RoboDK station: Assembly-with-ABB-IRB-2400-16.rdk

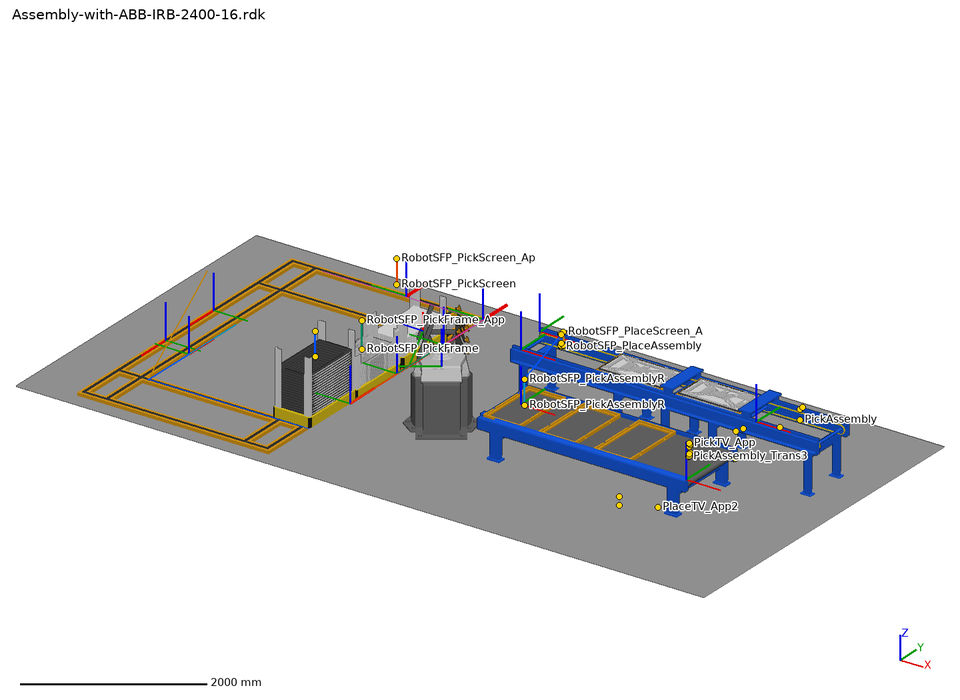
[picture v0: the station drawn from its stored meshes, robots at their saved joint values, targets as dots, program paths as lines]
Station Assembly with ABB IRB 2400/16 (saved by RoboDK 5.6.8). Poses are relative to the parent item; angles as X-Y-Z fixed-axis rotations.
Station parameters (name, value as stored): Assembly, 1, NextAssembly, 1, ScrewCircuit, 1, BuildCircuit, 1, UpFoamDone, 0, RackReady, 0, TAGS, ['Assembly']
  - folder First_Assembly_Station
    - folder Python
      - Python program RackConveyor_Next (listed below)
      - Python program MainConveyor_Next (listed below)
    - folder RobotSFP_Programs
      - folder Gripper1
        - program Gripper1Open (2 instructions, listed below)
        - program Gripper1CloseFrame (2 instructions, listed below)
        - program Gripper1CloseAssemRack (2 instructions, listed below)
        - program Gripper1OpenPartial (2 instructions, listed below)
        - program Gripper1CloseFrontPanel (2 instructions, listed below)
      - folder AssemblyPicks
        - program PickFrontPanel (8 instructions, listed below)
        - program PickScreen (6 instructions, listed below)
        - program PickFrame (8 instructions, listed below)
      - folder PlaceOnAssembly
        - program PlaceFrontPanel (9 instructions, listed below)
        - program PlaceScreen (9 instructions, listed below)
        - program PickAndPlace_AssemRack (14 instructions, listed below)
        - program PlaceFrame (11 instructions, listed below)
      - folder AssemblyProcess
        - program AssemblyTV (6 instructions, listed below)
    - frame MainConveyor Base at (-1580, 450, 650) mm
      - robot MainConveyor: 1 axes
          modified DH rows (alpha deg, a mm, theta deg, d mm): 0, 0, 0, 0 linear
          base shift (0, 0, 0) mm, rotated rx 0 ry 90 rz 0 deg
          joint limits [-200000] to [200000]; home [0]; saved at [0]
        - frame MainConveyorRef at (90, -480, 0) mm
          - object TVAssemblies at (2875, 462, 0) mm, rotated rx 0 ry 0 rz -180 deg, size 1893 x 485 x 64 mm
      - frame MainConveyorRef_Init at (3165, -480, 0) mm
        - object TVAssemblies at (-200, 462, 0) mm, rotated rx 0 ry 0 rz -180 deg, size 1893 x 485 x 64 mm
      - frame RobotSFP_Targets at (-1430, 980, -645) mm, rotated rx 0 ry 0 rz 90 deg
        - frame AssemblyRack_Targets at (0, 1000, 0) mm
          - target RobotSFP_PickAssemblyRack (Cartesian target) at (-2266, -3132, 478) mm, rotated rx 180 ry 0 rz -180 deg; joints [-130.241, 56.24, 97.421, -5.047, -77.391, -90.693] of ABB IRB 2400/16
          - target RobotSFP_PickAssemblyRack_App (Cartesian target) at (-2266, -3132, 790) mm, rotated rx -180 ry 0 rz -180 deg; joints [-130.241, 25.611, 75.665, -5.962, -55.732, -88.432] of ABB IRB 2400/16
          - target RobotSFP_PlaceAssemblyRack (Cartesian target) at (-1226, -2885, 690) mm, rotated rx 180 ry 0 rz -90 deg; joints [-92.609, 47.662, 66.312, -67.815, -58.973, -66.679] of ABB IRB 2400/16
          - target RobotSFP_PlaceAssemblyRack_App (Cartesian target) at (-1226, -2885, 830) mm, rotated rx -180 ry 0 rz -90 deg; joints [-92.609, 38.532, 58.57, -72.434, -56.335, -58.059] of ABB IRB 2400/16
        - frame TvAssembly at (0, 0, -20) mm
          - target RobotSFP_PlaceFrontPanel (Cartesian target) at (-1232.5, -1885.5, 730.48) mm, rotated rx 180 ry 0 rz -90 deg; joints [-92.924, 46.128, 65.422, -68.631, -58.762, -65.657] of ABB IRB 2400/16
          - target RobotSFP_PlaceFrontPanel_App (Cartesian target) at (-1232.5, -1885.5, 863.5) mm, rotated rx -180 ry 0 rz -90 deg; joints [-92.924, 37.534, 57.905, -73.159, -56.297, -57.237] of ABB IRB 2400/16
          - target RobotSFP_PlaceScreen (Cartesian target) at (-1189.8, -1890.5, 709.68) mm, rotated rx 180 ry 0 rz 90 deg; joints [-91.494, 45.247, 62.599, -68.849, -57.154, 117.178] of ABB IRB 2400/16
          - target RobotSFP_PlaceScreen_App (Cartesian target) at (-1189.8, -1890.5, 871.7) mm, rotated rx 180 ry 0 rz 90 deg; joints [-91.494, 35.396, 53.282, -74.906, -54.246, 127.901] of ABB IRB 2400/16
          - target RobotSFP_PlaceFrame (Cartesian target) at (-1219.5, -1885.2, 745.48) mm, rotated rx 180 ry 0 rz -90 deg; joints [-92.315, 45.44, 64.267, -68.683, -58.101, -64.505] of ABB IRB 2400/16
          - target RobotSFP_PlaceFrame_App (Cartesian target) at (-1219.5, -1885.2, 853.5) mm, rotated rx -180 ry 0 rz -90 deg; joints [-92.315, 38.518, 58.189, -72.396, -56.073, -57.678] of ABB IRB 2400/16
      - frame PickAssembly_Targets at (89.8, -480, -648) mm
        - target PickAssembly (Cartesian target) at (3485.2, 228, 693.7) mm, rotated rx -180 ry 0 rz -180 deg; joints [22.371, 48.063, -2.442, 0, 44.379, 112.371]
        - target PickAssembly_App (Cartesian target) at (3485.2, 228, 823.7) mm, rotated rx -180 ry 0 rz -180 deg; joints [22.371, 43.327, -4.321, 0, 50.994, 112.371]
        - target PickAssembly_Trans1 (Cartesian target) at (3525.2, 228, 853.7) mm, rotated rx 180 ry 5 rz 180 deg; joints [21.562, 41.902, -4.058, -5.74, 54.134, 115.007]
        - target PickAssembly_Trans2 (Cartesian target) at (3605.2, -312, 853.7) mm, rotated rx -180 ry 0 rz 80 deg; joints [28.286, 14.78, 41.406, 0, 33.814, 218.286]
        - target PickAssembly_Trans3 (Cartesian target) at (2776, -836.2, 483.7) mm, rotated rx -180 ry 0 rz 90 deg; joints [77.346, 50.715, 13.544, 0, 25.741, 257.346]
      - object Floor at (-100, -970, -650) mm, size 9000 x 4500 x 0 mm, geometry from Floor (2).sld
    - frame ABB IRB 2400/16 Base at (-2010, -770, 600) mm, rotated rx 0 ry 0 rz 125 deg
      - robot ABB IRB 2400/16: 6 axes, payload 16 kg, reach 1550 mm, repeatability 0.03 mm, weight 380 kg
          joint limits [-180, -100, -60, -200, -120, -400] to [180, 110, 65, 200, 120, 400]; home [0, 0, 0, 0, 0, 0]; saved at [-92.609, 38.532, 58.57, -72.434, -56.335, -58.059]
        - frame ToolRobot1 Base at (0, 195, 425) mm, rotated rx -70 ry 0 rz 0 deg
          - robot ToolRobot1: 1 axes
              joint limits [-20] to [200]; home [0]; saved at [26]
        - tool ToolRobot1_TCP_Gripper, TCP at (0, 195, 425) mm, rotated rx -70 ry 0 rz 0 deg
        - tool ToolRobot1_TCP_Cup, TCP at (0, -240, 450) mm, rotated rx 70 ry 0 rz 0 deg
      - target Gripper1Open (Cartesian target) at (1586.9, 365.98, 80) mm, rotated rx 180 ry 0 rz -35 deg; joints [100, -0.574, 0, 0, -0.574, -0.819] of ToolRobot1
      - target Gripper1CloseFrame (Cartesian target) at (858.67, 851.47, -365) mm, rotated rx -180 ry 0 rz -35 deg; joints [-4, 0, 0, 0, 0, 0] of ToolRobot1
      - target Gripper1CloseAssemRack (Cartesian target) at (-703.35, -889.42, -270) mm, rotated rx 180 ry 0 rz 145 deg; joints [26, 0.574, 0, 0, 0.574, 0.819] of ToolRobot1
      - target Gripper1OpenPartial (Cartesian target) at (320.55, -1292.63, -60) mm, rotated rx -180 ry 0 rz -125 deg; joints [50, -0.819, 0, 0, -0.819, 0.574] of ToolRobot1
      - target Gripper1CloseFrontPanel (Cartesian target) at (136.59, 1363.18, -105) mm, rotated rx -180 ry 0 rz -35 deg; joints [41, -0.574, 0, 0, -0.574, -0.819] of ToolRobot1
      - object Robot1_Stand at (0, 0, 0) mm, size 938.8 x 824.6 x 600 mm, geometry from Robot1_Stand.step
    - frame AssemblyRackConveyor Base at (1530, -1260, 440) mm
      - robot AssemblyRackConveyor: 1 axes
          modified DH rows (alpha deg, a mm, theta deg, d mm): 0, 0, 0, 0 linear
          base shift (0, 0, 0) mm, rotated rx 0 ry 90 rz 0 deg
          joint limits [-200000] to [200000]; home [0]; saved at [0]
        - frame AssemblyRackConveyorRef at (0, 0, 0) mm
          - object AssemblyRack at (-1440, 0, 0) mm, size 40 x 853 x 485 mm, geometry from AssemblyRack.step
          - object AssemblyRack at (-720, 0, 0) mm, size 40 x 853 x 485 mm, geometry from AssemblyRack.step
          - object AssemblyRack at (-2160, 0, 0) mm, size 40 x 853 x 485 mm, geometry from AssemblyRack.step
      - frame AssemblyRackConveyorRef_Init at (0, 0, 0) mm
        - object AssemblyRack_Ref at (-1440, 0, 0) mm, size 40 x 853 x 485 mm, geometry from AssemblyRack.step
        - object AssemblyRack_Ref at (-720, 0, 0) mm, size 40 x 853 x 485 mm, geometry from AssemblyRack.step
        - object AssemblyRack_Ref at (-2160, 0, 0) mm, size 40 x 853 x 485 mm, geometry from AssemblyRack.step
      - frame AssemblyRackConveyor_Targets at (0, 0, 0) mm
        - target PlaceAssembly_App1 (Cartesian target) at (509.67, 338.93, 613.53) mm, rotated rx -172.41 ry 0.65 rz 63.37 deg; joints [68.32, -23.6, 57.9, -0.01, 48.08, 275]
        - target PlaceAssembly (Cartesian target) at (-254, 423.8, 43.7) mm, rotated rx -180 ry 0 rz 90 deg; joints [77.346, 50.715, 13.544, 0, 25.741, 257.346]
        - target PlaceAssembly_App2 (Cartesian target) at (-254, 423.8, 153.7) mm, rotated rx 180 ry 0 rz 90 deg; joints [77.346, 45.066, 13.905, -180, -31.029, 77.346]
        - target PlaceBackPanel (Cartesian target) at (-241, 423.9, 86) mm, rotated rx 180 ry 0 rz -90 deg; joints [77.214, 48.026, 14.946, 0, 27.028, 77.214]
        - target PlaceBackPanel_App1 (Cartesian target) at (481.6, 244.34, 613.6) mm, rotated rx 172.37 ry 0 rz -101.17 deg; joints [78.83, -23.59, 57.89, 0, 48.07, 90]
        - target PickTV (Cartesian target) at (-252, 423.9, 65) mm, rotated rx 180 ry 0 rz -90 deg; joints [77.322, 49.521, 13.865, 0, 26.614, 77.322]
        - target PlaceBackPanel_App2 (Cartesian target) at (-241, 423.9, 176) mm, rotated rx 180 ry 0 rz -90 deg; joints [77.214, 43.448, 15.011, 0, 31.541, 77.214]
        - target PickTV_App (Cartesian target) at (-252, 423.9, 195) mm, rotated rx 180 ry 0 rz -90 deg; joints [77.322, 42.97, 13.968, 0, 33.062, 77.322]
        - target PlaceTV_App1 (Cartesian target) at (349, 423.9, 176) mm, rotated rx 180 ry 0 rz -90 deg; joints [66.756, 24.897, 59.615, 0, 5.488, 66.756]
        - target PlaceTV_App2 (Cartesian target) at (349, -1026.1, 176) mm, rotated rx -180 ry 0 rz -90 deg; joints [150.453, 45.871, 9.692, 0, 34.437, 150.453]
        - target PlaceTV (Cartesian target) at (-141, -1045, 72) mm, rotated rx 180 ry 0 rz -90 deg; joints [135.834, 66.25, -25.615, 0, 49.365, 135.834]
        - target PlaceTV_App3 (Cartesian target) at (-141, -1045, 172) mm, rotated rx -180 ry 0 rz -90 deg; joints [135.834, 62.358, -25.443, 0, 53.085, 135.834]
    - program TVAssembly_Main (5 instructions, listed below)
  - folder AVG_On_Rail
    - folder Python
      - Python program Next_RackTarget (listed below)
    - folder TvRack_Programs
      - program TvRack_ToPickUp (5 instructions, listed below)
      - program TvRack_FrontPanel_ToPickUp (4 instructions, listed below)
      - program TvRack_Frame_ToPickUp (4 instructions, listed below)
      - program TvRack_Screen_ToPickUp (4 instructions, listed below)
      - program TvRack_BackToFill (5 instructions, listed below)
      - program TvRack_FrontPanel_ToFill (4 instructions, listed below)
      - program TvRack_Frame_ToFill (4 instructions, listed below)
      - program TvRack_Screen_ToFill (4 instructions, listed below)
    - frame TvRack_Rail at (-3000, 1420, 0) mm, rotated rx 0 ry 0 rz 90 deg
      - robot TvRack_FrontPanel: 2 axes
          modified DH rows (alpha deg, a mm, theta deg, d mm): 0, 0, 0, 0 linear; 90, 0, 0, 0 linear
          base shift (0, 0, 0) mm, rotated rx 0 ry 90 rz 0 deg
          joint limits [-3250, -2100] to [0, 0]; home [0, 0]; saved at [-2480, 0]
        - frame TvRack_FrontPanel_Ref at (0, 0, 0) mm
          - object TVFrontPanel at (-750, 400, 0) mm, rotated rx 0 ry 0 rz 180 deg, size 812.6 x 460.3 x 32.5 mm, geometry from TVFrontCase.step
          - object TVFrontPanel at (-750, 400, 30) mm, rotated rx 0 ry 0 rz 180 deg, size 812.6 x 460.3 x 32.5 mm, geometry from TVFrontCase.step
          - object TVFrontPanel at (-750, 400, 60) mm, rotated rx 0 ry 0 rz 180 deg, size 812.6 x 460.3 x 32.5 mm, geometry from TVFrontCase.step
          - object TVFrontPanel at (-750, 400, 90) mm, rotated rx 0 ry 0 rz 180 deg, size 812.6 x 460.3 x 32.5 mm, geometry from TVFrontCase.step
          - object TVFrontPanel at (-750, 400, 120) mm, rotated rx 0 ry 0 rz 180 deg, size 812.6 x 460.3 x 32.5 mm, geometry from TVFrontCase.step
          - object TVFrontPanel at (-750, 400, 150) mm, rotated rx 0 ry 0 rz 180 deg, size 812.6 x 460.3 x 32.5 mm, geometry from TVFrontCase.step
          - object TVFrontPanel at (-750, 400, 180) mm, rotated rx 0 ry 0 rz 180 deg, size 812.6 x 460.3 x 32.5 mm, geometry from TVFrontCase.step
          - object TVFrontPanel at (-750, 400, 210) mm, rotated rx 0 ry 0 rz 180 deg, size 812.6 x 460.3 x 32.5 mm, geometry from TVFrontCase.step
          - object TVFrontPanel at (-750, 400, 270) mm, rotated rx 0 ry 0 rz 180 deg, size 812.6 x 460.3 x 32.5 mm, geometry from TVFrontCase.step
          - object TVFrontPanel at (-750, 400, 240) mm, rotated rx 0 ry 0 rz 180 deg, size 812.6 x 460.3 x 32.5 mm, geometry from TVFrontCase.step
          - object TVFrontPanel at (-750, 400, 300) mm, rotated rx 0 ry 0 rz 180 deg, size 812.6 x 460.3 x 32.5 mm, geometry from TVFrontCase.step
          - object TVFrontPanel at (-750, 400, 330) mm, rotated rx 0 ry 0 rz 180 deg, size 812.6 x 460.3 x 32.5 mm, geometry from TVFrontCase.step
          - object TVFrontPanel at (-750, 400, 360) mm, rotated rx 0 ry 0 rz 180 deg, size 812.6 x 460.3 x 32.5 mm, geometry from TVFrontCase.step
          - object TVFrontPanel at (-750, 400, 390) mm, rotated rx 0 ry 0 rz 180 deg, size 812.6 x 460.3 x 32.5 mm, geometry from TVFrontCase.step
          - object TVFrontPanel at (-750, 400, 420) mm, rotated rx 0 ry 0 rz 180 deg, size 812.6 x 460.3 x 32.5 mm, geometry from TVFrontCase.step
          - object TVFrontPanel at (-750, 400, 450) mm, rotated rx 0 ry 0 rz 180 deg, size 812.6 x 460.3 x 32.5 mm, geometry from TVFrontCase.step
      - robot TvRack_Frame: 2 axes
          modified DH rows (alpha deg, a mm, theta deg, d mm): 0, 0, 0, 0 linear; 90, 0, 0, 0 linear
          base shift (0, 0, 0) mm, rotated rx 0 ry 90 rz 0 deg
          joint limits [-3250, -2100] to [0, 0]; home [0, 0]; saved at [-1600, 0]
        - frame TvRack_Frame_Ref at (0, 0, 0) mm
          - object TVFrame at (-750, 400, 0) mm, rotated rx 0 ry 0 rz -180 deg, size 786.6 x 406 x 28 mm, geometry from TVFrame.step
          - object TVFrame at (-750, 400, 15) mm, rotated rx 0 ry 0 rz -180 deg, size 786.6 x 406 x 28 mm, geometry from TVFrame.step
          - object TVFrame at (-750, 400, 30) mm, rotated rx 0 ry 0 rz -180 deg, size 786.6 x 406 x 28 mm, geometry from TVFrame.step
          - object TVFrame at (-750, 400, 45) mm, rotated rx 0 ry 0 rz -180 deg, size 786.6 x 406 x 28 mm, geometry from TVFrame.step
          - object TVFrame at (-750, 400, 60) mm, rotated rx 0 ry 0 rz -180 deg, size 786.6 x 406 x 28 mm, geometry from TVFrame.step
          - object TVFrame at (-750, 400, 75) mm, rotated rx 0 ry 0 rz -180 deg, size 786.6 x 406 x 28 mm, geometry from TVFrame.step
          - object TVFrame at (-750, 400, 90) mm, rotated rx 0 ry 0 rz -180 deg, size 786.6 x 406 x 28 mm, geometry from TVFrame.step
          - object TVFrame at (-750, 400, 105) mm, rotated rx 0 ry 0 rz -180 deg, size 786.6 x 406 x 28 mm, geometry from TVFrame.step
          - object TVFrame at (-750, 400, 120) mm, rotated rx 0 ry 0 rz -180 deg, size 786.6 x 406 x 28 mm, geometry from TVFrame.step
          - object TVFrame at (-750, 400, 135) mm, rotated rx 0 ry 0 rz -180 deg, size 786.6 x 406 x 28 mm, geometry from TVFrame.step
          - object TVFrame at (-750, 400, 225) mm, rotated rx 0 ry 0 rz -180 deg, size 786.6 x 406 x 28 mm, geometry from TVFrame.step
          - object TVFrame at (-750, 400, 210) mm, rotated rx 0 ry 0 rz -180 deg, size 786.6 x 406 x 28 mm, geometry from TVFrame.step
          - object TVFrame at (-750, 400, 195) mm, rotated rx 0 ry 0 rz -180 deg, size 786.6 x 406 x 28 mm, geometry from TVFrame.step
          - object TVFrame at (-750, 400, 180) mm, rotated rx 0 ry 0 rz -180 deg, size 786.6 x 406 x 28 mm, geometry from TVFrame.step
          - object TVFrame at (-750, 400, 165) mm, rotated rx 0 ry 0 rz -180 deg, size 786.6 x 406 x 28 mm, geometry from TVFrame.step
          - object TVFrame at (-750, 400, 150) mm, rotated rx 0 ry 0 rz -180 deg, size 786.6 x 406 x 28 mm, geometry from TVFrame.step
      - robot TvRack_Screen: 2 axes
          modified DH rows (alpha deg, a mm, theta deg, d mm): 0, 0, 0, 0 linear; 90, 0, 0, 0 linear
          base shift (0, 0, 0) mm, rotated rx 0 ry 90 rz 0 deg
          joint limits [-3250, -2100] to [0, 0]; home [0, 0]; saved at [-730, 0]
        - frame TvRack_Screen_Ref at (0, 0, 0) mm
          - object TVScreen at (0, 0, 0) mm, size 776.6 x 396 x 12 mm, geometry from TVScreen.step
          - object TVScreen at (0, 0, 12) mm, size 776.6 x 396 x 12 mm, geometry from TVScreen.step
          - object TVScreen at (0, 0, 24) mm, size 776.6 x 396 x 12 mm, geometry from TVScreen.step
          - object TVScreen at (0, 0, 36) mm, size 776.6 x 396 x 12 mm, geometry from TVScreen.step
          - object TVScreen at (0, 0, 48) mm, size 776.6 x 396 x 12 mm, geometry from TVScreen.step
          - object TVScreen at (0, 0, 60) mm, size 776.6 x 396 x 12 mm, geometry from TVScreen.step
          - object TVScreen at (0, 0, 72) mm, size 776.6 x 396 x 12 mm, geometry from TVScreen.step
          - object TVScreen at (0, 0, 84) mm, size 776.6 x 396 x 12 mm, geometry from TVScreen.step
          - object TVScreen at (0, 0, 96) mm, size 776.6 x 396 x 12 mm, geometry from TVScreen.step
          - object TVScreen at (0, 0, 108) mm, size 776.6 x 396 x 12 mm, geometry from TVScreen.step
          - object TVScreen at (0, 0, 120) mm, size 776.6 x 396 x 12 mm, geometry from TVScreen.step
          - object TVScreen at (0, 0, 132) mm, size 776.6 x 396 x 12 mm, geometry from TVScreen.step
          - object TVScreen at (0, 0, 144) mm, size 776.6 x 396 x 12 mm, geometry from TVScreen.step
          - object TVScreen at (0, 0, 180) mm, size 776.6 x 396 x 12 mm, geometry from TVScreen.step
          - object TVScreen at (0, 0, 168) mm, size 776.6 x 396 x 12 mm, geometry from TVScreen.step
          - object TVScreen at (0, 0, 156) mm, size 776.6 x 396 x 12 mm, geometry from TVScreen.step
      - frame TvRack_FrontPanel_Init at (-1460, 2500, 0) mm, rotated rx 0 ry 0 rz 180 deg
        - object TVFrontPanel_Ref at (0, 0, 0) mm, size 812.6 x 460.3 x 32.5 mm, geometry from TVFrontCase.step
        - object TVFrontPanel_Ref at (0, 0, 30) mm, size 812.6 x 460.3 x 32.5 mm, geometry from TVFrontCase.step
        - object TVFrontPanel_Ref at (0, 0, 60) mm, size 812.6 x 460.3 x 32.5 mm, geometry from TVFrontCase.step
        - object TVFrontPanel_Ref at (0, 0, 90) mm, size 812.6 x 460.3 x 32.5 mm, geometry from TVFrontCase.step
        - object TVFrontPanel_Ref at (0, 0, 120) mm, size 812.6 x 460.3 x 32.5 mm, geometry from TVFrontCase.step
        - object TVFrontPanel_Ref at (0, 0, 150) mm, size 812.6 x 460.3 x 32.5 mm, geometry from TVFrontCase.step
        - object TVFrontPanel_Ref at (0, 0, 180) mm, size 812.6 x 460.3 x 32.5 mm, geometry from TVFrontCase.step
        - object TVFrontPanel_Ref at (0, 0, 210) mm, size 812.6 x 460.3 x 32.5 mm, geometry from TVFrontCase.step
        - object TVFrontPanel_Ref at (0, 0, 270) mm, size 812.6 x 460.3 x 32.5 mm, geometry from TVFrontCase.step
        - object TVFrontPanel_Ref at (0, 0, 240) mm, size 812.6 x 460.3 x 32.5 mm, geometry from TVFrontCase.step
        - object TVFrontPanel_Ref at (0, 0, 300) mm, size 812.6 x 460.3 x 32.5 mm, geometry from TVFrontCase.step
        - object TVFrontPanel_Ref at (0, 0, 330) mm, size 812.6 x 460.3 x 32.5 mm, geometry from TVFrontCase.step
        - object TVFrontPanel_Ref at (0, 0, 360) mm, size 812.6 x 460.3 x 32.5 mm, geometry from TVFrontCase.step
        - object TVFrontPanel_Ref at (0, 0, 390) mm, size 812.6 x 460.3 x 32.5 mm, geometry from TVFrontCase.step
        - object TVFrontPanel_Ref at (0, 0, 420) mm, size 812.6 x 460.3 x 32.5 mm, geometry from TVFrontCase.step
        - object TVFrontPanel_Ref at (0, 0, 450) mm, size 812.6 x 460.3 x 32.5 mm, geometry from TVFrontCase.step
      - frame TvRack_Frame_Init at (-2350, 2500, 0) mm, rotated rx 0 ry 0 rz -180 deg
        - object TVFrame_Ref at (0, 0, 0) mm, size 786.6 x 406 x 28 mm, geometry from TVFrame.step
        - object TVFrame_Ref at (0, 0, 15) mm, size 786.6 x 406 x 28 mm, geometry from TVFrame.step
        - object TVFrame_Ref at (0, 0, 30) mm, size 786.6 x 406 x 28 mm, geometry from TVFrame.step
        - object TVFrame_Ref at (0, 0, 45) mm, size 786.6 x 406 x 28 mm, geometry from TVFrame.step
        - object TVFrame_Ref at (0, 0, 60) mm, size 786.6 x 406 x 28 mm, geometry from TVFrame.step
        - object TVFrame_Ref at (0, 0, 75) mm, size 786.6 x 406 x 28 mm, geometry from TVFrame.step
        - object TVFrame_Ref at (0, 0, 90) mm, size 786.6 x 406 x 28 mm, geometry from TVFrame.step
        - object TVFrame_Ref at (0, 0, 105) mm, size 786.6 x 406 x 28 mm, geometry from TVFrame.step
        - object TVFrame_Ref at (0, 0, 120) mm, size 786.6 x 406 x 28 mm, geometry from TVFrame.step
        - object TVFrame_Ref at (0, 0, 135) mm, size 786.6 x 406 x 28 mm, geometry from TVFrame.step
        - object TVFrame_Ref at (0, 0, 225) mm, size 786.6 x 406 x 28 mm, geometry from TVFrame.step
        - object TVFrame_Ref at (0, 0, 210) mm, size 786.6 x 406 x 28 mm, geometry from TVFrame.step
        - object TVFrame_Ref at (0, 0, 195) mm, size 786.6 x 406 x 28 mm, geometry from TVFrame.step
        - object TVFrame_Ref at (0, 0, 180) mm, size 786.6 x 406 x 28 mm, geometry from TVFrame.step
        - object TVFrame_Ref at (0, 0, 165) mm, size 786.6 x 406 x 28 mm, geometry from TVFrame.step
        - object TVFrame_Ref at (0, 0, 150) mm, size 786.6 x 406 x 28 mm, geometry from TVFrame.step
      - frame TvRack_Screen_Init at (-2480, 2100, 0) mm
        - object TVScreen_Ref at (0, 0, 0) mm, size 776.6 x 396 x 12 mm, geometry from TVScreen.step
        - object TVScreen_Ref at (0, 0, 12) mm, size 776.6 x 396 x 12 mm, geometry from TVScreen.step
        - object TVScreen_Ref at (0, 0, 24) mm, size 776.6 x 396 x 12 mm, geometry from TVScreen.step
        - object TVScreen_Ref at (0, 0, 36) mm, size 776.6 x 396 x 12 mm, geometry from TVScreen.step
        - object TVScreen_Ref at (0, 0, 48) mm, size 776.6 x 396 x 12 mm, geometry from TVScreen.step
        - object TVScreen_Ref at (0, 0, 60) mm, size 776.6 x 396 x 12 mm, geometry from TVScreen.step
        - object TVScreen_Ref at (0, 0, 72) mm, size 776.6 x 396 x 12 mm, geometry from TVScreen.step
        - object TVScreen_Ref at (0, 0, 84) mm, size 776.6 x 396 x 12 mm, geometry from TVScreen.step
        - object TVScreen_Ref at (0, 0, 96) mm, size 776.6 x 396 x 12 mm, geometry from TVScreen.step
        - object TVScreen_Ref at (0, 0, 108) mm, size 776.6 x 396 x 12 mm, geometry from TVScreen.step
        - object TVScreen_Ref at (0, 0, 120) mm, size 776.6 x 396 x 12 mm, geometry from TVScreen.step
        - object TVScreen_Ref at (0, 0, 132) mm, size 776.6 x 396 x 12 mm, geometry from TVScreen.step
        - object TVScreen_Ref at (0, 0, 144) mm, size 776.6 x 396 x 12 mm, geometry from TVScreen.step
        - object TVScreen_Ref at (0, 0, 180) mm, size 776.6 x 396 x 12 mm, geometry from TVScreen.step
        - object TVScreen_Ref at (0, 0, 168) mm, size 776.6 x 396 x 12 mm, geometry from TVScreen.step
        - object TVScreen_Ref at (0, 0, 156) mm, size 776.6 x 396 x 12 mm, geometry from TVScreen.step
      - frame TvRack_Targets at (0, 0, 0) mm
        - frame TvRack_Frame_Targets at (0, 0, 0) mm
          - target TvRack_Frame_Go2 (Cartesian target) at (0, 0, 0) mm; joints [0, 0, 0, 0, 0, 1] of TvRack_Frame
          - target TvRack_Frame_GoPickUp (Cartesian target) at (-1600, 0, 0) mm; joints [-1600, 0, 0, 0, 0, 1] of TvRack_Frame
          - target TvRack_Frame_Go3 (Cartesian target) at (-3250, 0, 0) mm; joints [-3250, 0, 0, 0, 0, 0] of TvRack_Frame
          - target TvRack_Frame_Go4 (Cartesian target) at (-3250, 2100, 0) mm; joints [-3250, -2100, 0, 0, 0, 1] of TvRack_Frame
          - target TvRack_Frame_Go1 (Cartesian target) at (0, 2100, 0) mm; joints [0, -2100, 0, 0, 0, 0] of TvRack_Frame
          - target TvRack_Frame_Fill (Cartesian target) at (-1600, 2100, 0) mm; joints [-1600, -2100, 0, 0, 0, 0] of TvRack_Frame
        - frame TvRack_Screen_Targets at (0, 0, 0) mm
          - target TvRack_Screen_Go1 (Cartesian target) at (0, 2100, 0) mm; joints [0, -2100, 0, 0, 0, 0] of TvRack_Screen
          - target TvRack_Screen_Fill (Cartesian target) at (-2480, 2100, 0) mm; joints [-2480, -2100, 0, 0, 0, 0] of TvRack_Screen
          - target TvRack_Screen_Go2 (Cartesian target) at (0, 0, 0) mm; joints [0, 0, 0, 0, 0, 0] of TvRack_Screen
          - target TvRack_Screen_GoPickUp (Cartesian target) at (-730, 0, 0) mm; joints [-730, 0, 0, 0, 0, 0] of TvRack_Screen
          - target TvRack_Screen_Go3 (Cartesian target) at (-3250, 0, 0) mm; joints [-3250, 0, 0, 0, 0, 0] of TvRack_Screen
          - target TvRack_Screen_Go4 (Cartesian target) at (-3250, 2100, 0) mm; joints [-3250, -2100, 0, 0, 0, 0] of TvRack_Screen
        - frame TvRack_FrontPanel_Targets at (0, 1000, 0) mm
          - target TvRack_FrontPanel_Go1 (Cartesian target) at (0, 1100, 0) mm; joints [0, -2100, 0, 0, 0, 0] of TvRack_FrontPanel
          - target TvRack_FrontPanel_Fill (Cartesian target) at (-710, 2100, 0) mm; joints [-710, -2100, 0, 0, 0, 0] of TvRack_FrontPanel
          - target TvRack_FrontPanel_Go2 (Cartesian target) at (0, -1000, 0) mm; joints [0, 0, 0, 0, 0, 0] of TvRack_FrontPanel
          - target TvRack_FrontPanel_GoPickUp (Cartesian target) at (-2480, -1000, 0) mm; joints [-2480, 0, 0, 0, 0, 0] of TvRack_FrontPanel
          - target TvRack_FrontPanel_Go3 (Cartesian target) at (-3250, -1000, 0) mm; joints [-3250, 0, 0, 0, 0, 0] of TvRack_FrontPanel
          - target TvRack_FrontPanel_Go4 (Cartesian target) at (-3250, 1100, 0) mm; joints [-3250, -2100, 0, 0, 0, 0] of TvRack_FrontPanel
      - frame RobotSFP_Targets at (0, 0, 0) mm
        - frame RobotSFP_Targets_Screen at (-730, 0, 0) mm
          - target RobotSFP_PickScreen_App (Cartesian target) at (-370, 355, 1070) mm, rotated rx 40 ry 0 rz -180 deg; joints [1.245, 64.461, 46.78, -77.31, -50.972, 135.312] of ABB IRB 2400/16
          - target RobotSFP_PickScreen (Cartesian target) at (-370, 355, 767) mm, rotated rx 40 ry 0 rz -180 deg; joints [1.245, 83.731, 54.243, -71.676, -52.972, 126.179] of ABB IRB 2400/16
        - frame RobotSFP_Targets_Frame at (-1600, 0, 0) mm
          - target RobotSFP_PickFrame_App (Cartesian target) at (-375, 200, 725) mm, rotated rx -180 ry 0 rz 0 deg; joints [39.541, 35.433, 77.282, -17.219, -57.79, -86.023] of ABB IRB 2400/16
          - target RobotSFP_PickFrame (Cartesian target) at (-375, 200, 389) mm, rotated rx -180 ry 0 rz 0 deg; joints [39.541, 65.197, 95.152, -15.031, -74.971, -91.42] of ABB IRB 2400/16
        - frame RobotSFP_Targets_FrontPanel at (-2480, 0, 0) mm
          - target RobotSFP_PickFrontPanel (Cartesian target) at (-375, 193, 654) mm, rotated rx -180 ry 0 rz 0 deg; joints [95.799, 49.208, 70.093, 48.023, -55.681, -105.627] of ABB IRB 2400/16
          - target RobotSFP_PickFrontPanel_App (Cartesian target) at (-375, 193, 955) mm, rotated rx -180 ry 0 rz 0 deg; joints [95.799, 29.69, 52.296, 60.06, -45.117, -124.332] of ABB IRB 2400/16
  - folder Reset_Scripts
    - Python program Reset_MainConveyor (listed below)
    - Python program Reset_Tool (listed below)
    - Python program Reset_RackConveyor (listed below)
    - Python program Render (listed below)
    - Python program Reset_AVG (listed below)
    - Python program Reset_RackTargetRel (listed below)
    - Python program Reset_RackTargetABS (listed below)
  - program ResetALL (7 instructions, listed below)
  - program Main (6 instructions, listed below)
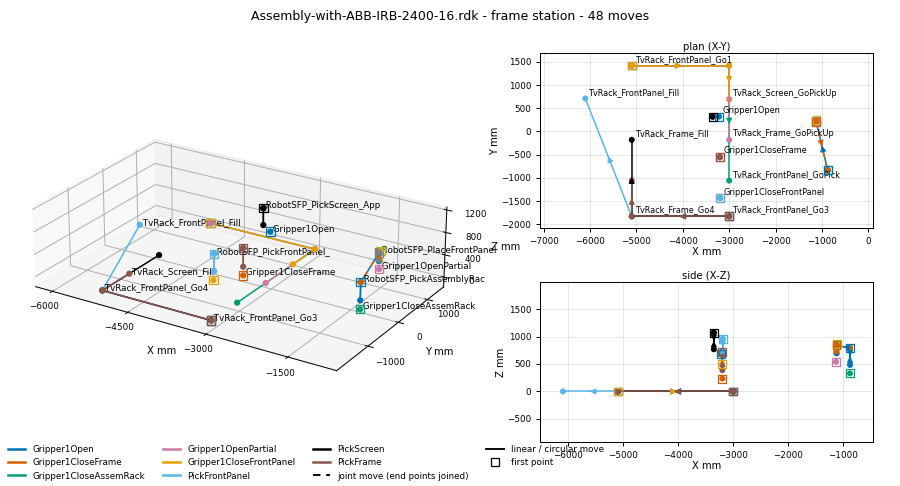
[picture p0: tool path of Assembly-with-ABB-IRB-2400-16.rdk in frame station, 48 of 48 moves have a stored position in this frame; points joined in program order, loops and branches not executed]

--- Python program RackConveyor_Next ---
# Type help("robolink") or help("robodk") for more information
# Press F5 to run the script
# Documentation: https://robodk.com/doc/en/RoboDK-API.html
# Reference:     https://robodk.com/doc/en/PythonAPI/index.html
# Note: It is not required to keep a copy of this file, your python script is saved with the station
from robodk import robolink
RDK = robolink.Robolink()

#----- Constants -----
MECHANISM_NAME = 'AssemblyRackConveyor'
PART_TRAVEL_MM = -720 #Travel for each box
NEW_REF_OBJECT_NAME = 'AssemblyRack_Ref' #Name of the ref object to copy
NEW_OBJECT_NAME = 'AssemblyRack' #Name of the new object created
REFERENCE_FRAME = 'AssemblyRackConveyorRef' #Name of the frame the object will move to
REFERENCE_FRAME_REF = 'AssemblyRackConveyorRef_Init'

#------- Program ------
mechanism = RDK.Item(MECHANISM_NAME,itemtype=robolink.ITEM_TYPE_ROBOT)
frame = RDK.Item(REFERENCE_FRAME, robolink.ITEM_TYPE_FRAME)
frame_ref = RDK.Item(REFERENCE_FRAME_REF, robolink.ITEM_TYPE_FRAME)
ref_obj = RDK.Item(NEW_REF_OBJECT_NAME, robolink.ITEM_TYPE_OBJECT)

if mechanism.Valid():
    mechanism.MoveJ(mechanism.Joints() + PART_TRAVEL_MM)

RDK.Render(False)

if mechanism.Valid():
    mechanism.setJoints([0])

if frame.Valid():
    for item in frame.Childs():
        if item.Type() == robolink.ITEM_TYPE_OBJECT:
            item.Delete()



for item in frame_ref.Childs():
    if frame.Valid() and  ref_obj.Valid():
        item.Copy()
        new_obj = RDK.Paste()
        new_obj.setVisible(False)
        new_obj.setParent(frame_ref)
        RDK.Update()
        new_obj.setName(NEW_OBJECT_NAME)
        new_obj.setParentStatic(frame)
        new_obj.setVisible(True)

RDK.Render(True)

--- Python program MainConveyor_Next ---
# Type help("robolink") or help("robodk") for more information
# Press F5 to run the script
# Documentation: https://robodk.com/doc/en/RoboDK-API.html
# Reference:     https://robodk.com/doc/en/PythonAPI/index.html
# Note: It is not required to keep a copy of this file, your python script is saved with the station
from robodk import robolink
RDK = robolink.Robolink()

#----- Constants -----
#---- Constant -----
NEW_REF_OBJECT_NAME = 'AssemblyRack_Ref' #Name of the ref object to copy
NEW_OBJECT_NAME = 'AssemblyRack' #Name of the new object created
REFERENCE_FRAME = 'MainConveyorRef' #Name of the frame the object will move to
REFERENCE_FRAME_REF = 'MainConveyorRef_Init'
MECHANISM_NAME = 'MainConveyor'
PART_TRAVEL_MM = -1040 #Travel

#------- Program ------
mechanism = RDK.Item(MECHANISM_NAME,itemtype=robolink.ITEM_TYPE_ROBOT)

if mechanism.Valid():
    mechanism.MoveJ(mechanism.Joints() + PART_TRAVEL_MM)


mechanism = RDK.Item(MECHANISM_NAME,itemtype=robolink.ITEM_TYPE_ROBOT)

#------- Program ------
frame = RDK.Item(REFERENCE_FRAME, robolink.ITEM_TYPE_FRAME)
frame_ref = RDK.Item(REFERENCE_FRAME_REF, robolink.ITEM_TYPE_FRAME)
ref_obj = RDK.Item(NEW_REF_OBJECT_NAME, robolink.ITEM_TYPE_OBJECT)


RDK.Render(False)

if mechanism.Valid():
    mechanism.setJoints([0])

if frame.Valid():
    for item in frame.Childs():
        if item.Type() == robolink.ITEM_TYPE_OBJECT:
            item.Delete()

for item in frame_ref.Childs():
    if frame.Valid() and  ref_obj.Valid():
        item.Copy()
        new_obj = RDK.Paste()
        new_obj.setVisible(False)
        new_obj.setParent(frame_ref)
        #new_obj.setName(NEW_OBJECT_NAME)
        RDK.Update()
        new_obj.setParentStatic(frame)
        new_obj.setVisible(True)

RDK.Render(True)

--- program Gripper1Open (robot ToolRobot1) ---
  Set Ref.: RobotSFP_Targets
  MoveJ (Gripper1Open)

--- program Gripper1CloseFrame (robot ToolRobot1) ---
  Set Ref.: RobotSFP_Targets
  MoveJ (Gripper1CloseFrame)

--- program Gripper1CloseAssemRack (robot ToolRobot1) ---
  Set Ref.: RobotSFP_Targets
  MoveJ (Gripper1CloseAssemRack)

--- program Gripper1OpenPartial (robot ToolRobot1) ---
  Set Ref.: RobotSFP_Targets
  MoveJ (Gripper1OpenPartial)

--- program Gripper1CloseFrontPanel (robot ToolRobot1) ---
  Set Ref.: RobotSFP_Targets
  MoveJ (Gripper1CloseFrontPanel)

--- program PickFrontPanel (robot ABB IRB 2400/16) ---
  Set Ref.: RobotSFP_Targets_FrontPanel
  Set Tool: ToolRobot1_TCP_Gripper
  Call Gripper1Open
  MoveJ (RobotSFP_PickFrontPanel_App)
  MoveL (RobotSFP_PickFrontPanel)
  Call Gripper1CloseFrontPanel
  Attach to ToolRobot1_TCP_Gripper
  MoveL (RobotSFP_PickFrontPanel_App)

--- program PickScreen (robot ABB IRB 2400/16) ---
  Set Ref.: RobotSFP_Targets_Screen
  Set Tool: ToolRobot1_TCP_Gripper
  MoveJ (RobotSFP_PickScreen_App)
  MoveL (RobotSFP_PickScreen)
  Attach to ToolRobot1_TCP_Cup
  MoveL (RobotSFP_PickScreen_App)

--- program PickFrame (robot ABB IRB 2400/16) ---
  Set Ref.: RobotSFP_Targets_Frame
  Set Tool: ToolRobot1_TCP_Gripper
  MoveJ (RobotSFP_PickFrame_App)
  Call Gripper1Open
  MoveL (RobotSFP_PickFrame)
  Call Gripper1CloseFrame
  Attach to ToolRobot1_TCP_Gripper
  MoveL (RobotSFP_PickFrame_App)

--- program PlaceFrontPanel (robot ABB IRB 2400/16) ---
  Set Ref.: TvAssembly
  Set Tool: ToolRobot1_TCP_Gripper
  MoveJ (RobotSFP_PlaceFrontPanel_App)
  Set speed (100.0 mm/s)
  MoveL (RobotSFP_PlaceFrontPanel)
  Call Gripper1OpenPartial
  Detach from ToolRobot1_TCP_Gripper
  Set speed (1000.0 mm/s)
  MoveJ (RobotSFP_PlaceFrontPanel_App)

--- program PlaceScreen (robot ABB IRB 2400/16) ---
  Set Ref.: TvAssembly
  Set Tool: ToolRobot1_TCP_Cup
  MoveJ (RobotSFP_PlaceScreen_App)
  Set speed (100.0 mm/s)
  MoveL (RobotSFP_PlaceScreen)
  Detach from ToolRobot1_TCP_Cup
  Pause 500 ms
  Set speed (1000.0 mm/s)
  MoveJ (RobotSFP_PlaceScreen_App)

--- program PickAndPlace_AssemRack (robot ABB IRB 2400/16) ---
  Set Ref.: AssemblyRack_Targets
  Call Gripper1Open
  Set Tool: ToolRobot1_TCP_Gripper
  MoveJ (RobotSFP_PickAssemblyRack_App)
  MoveL (RobotSFP_PickAssemblyRack)
  Call Gripper1CloseAssemRack
  Attach to ToolRobot1_TCP_Gripper
  MoveL (RobotSFP_PickAssemblyRack_App)
  MoveL (RobotSFP_PlaceAssemblyRack_App)
  MoveL (RobotSFP_PlaceAssemblyRack)
  Call Gripper1OpenPartial
  Detach from ToolRobot1_TCP_Gripper
  MoveL (RobotSFP_PlaceAssemblyRack_App)
  Call Gripper1Open

--- program PlaceFrame (robot ABB IRB 2400/16) ---
  Set Ref.: TvAssembly
  Set Tool: ToolRobot1_TCP_Gripper
  MoveJ (RobotSFP_PlaceFrame_App)
  Set speed (100.0 mm/s)
  MoveL (RobotSFP_PlaceFrame)
  Call Gripper1Open
  Detach from ToolRobot1_TCP_Gripper
  Set speed (1000.0 mm/s)
  MoveJ (RobotSFP_PlaceFrame_App)
  Set Ref.: AssemblyRack_Targets
  MoveJ (RobotSFP_PickAssemblyRack_App)

--- program AssemblyTV (robot ABB IRB 2400/16) ---
  Call PickFrontPanel
  Call PlaceFrontPanel
  Call PickScreen
  Call PlaceScreen
  Call PickFrame
  Call PlaceFrame

--- program TVAssembly_Main (robot ABB IRB 2400/16) ---
  Call PickAndPlace_AssemRack
  Call AssemblyTV
  Call Next_RackTarget
  Run RackConveyor_Next
  Call MainConveyor_Next

--- Python program Next_RackTarget ---
# Type help("robolink") or help("robodk") for more information
# Press F5 to run the script
# Documentation: https://robodk.com/doc/en/RoboDK-API.html
# Reference:     https://robodk.com/doc/en/PythonAPI/index.html
# Note: It is not required to keep a copy of this file, your python script is saved with the station
from robolink import *    # RoboDK API
from robodk import *      # Robot toolbox
RDK = Robolink()

#----- CONSTANT -----

TARGETscreen = 'RobotSFP_PickScreen'
TARGETframe = 'RobotSFP_PickFrame'
TARGETfrontpanel = 'RobotSFP_PickFrontPanel'
RDK.Render(False)

#----- PROGRAM -----
targetscreen = RDK.Item(TARGETscreen,ITEM_TYPE_TARGET)
targetfrontpanel = RDK.Item(TARGETfrontpanel,ITEM_TYPE_TARGET)
targetframe = RDK.Item(TARGETframe,ITEM_TYPE_TARGET)



targetscreen.setPose(Offset(targetscreen.Pose(),0,0,-12))
targetfrontpanel.setPose(Offset(targetfrontpanel.Pose(),0,0,-30))
targetframe.setPose(Offset(targetframe.Pose(),0,0,-15))

RDK.Render(True)
RDK.Update()

--- program TvRack_ToPickUp (robot TvRack_FrontPanel) ---
  Run TvRack_FrontPanel_ToPickUp
  Pause 1.0 s
  Run TvRack_Frame_ToPickUp
  Pause 1.0 s
  Call TvRack_Screen_ToPickUp

--- program TvRack_FrontPanel_ToPickUp (robot TvRack_FrontPanel) ---
  Set Ref.: TvRack_FrontPanel_Targets
  MoveL (TvRack_FrontPanel_Go1)
  MoveL (TvRack_FrontPanel_Go2)
  MoveL (TvRack_FrontPanel_GoPickUp)

--- program TvRack_Frame_ToPickUp (robot TvRack_Frame) ---
  Set Ref.: TvRack_Frame_Targets
  MoveL (TvRack_Frame_Go1)
  MoveL (TvRack_Frame_Go2)
  MoveL (TvRack_Frame_GoPickUp)

--- program TvRack_Screen_ToPickUp (robot TvRack_Screen) ---
  Set Ref.: TvRack_Screen_Targets
  MoveL (TvRack_Screen_Go1)
  MoveL (TvRack_Screen_Go2)
  MoveL (TvRack_Screen_GoPickUp)

--- program TvRack_BackToFill (robot TvRack_FrontPanel) ---
  Run TvRack_FrontPanel_ToFill
  Pause 1.0 s
  Run TvRack_Frame_ToFill
  Pause 1.0 s
  Call TvRack_Screen_ToFill

--- program TvRack_FrontPanel_ToFill (robot TvRack_FrontPanel) ---
  Set Ref.: TvRack_FrontPanel_Targets
  MoveL (TvRack_FrontPanel_Go3)
  MoveL (TvRack_FrontPanel_Go4)
  MoveL (TvRack_FrontPanel_Fill)

--- program TvRack_Frame_ToFill (robot TvRack_Frame) ---
  Set Ref.: TvRack_Frame_Targets
  MoveL (TvRack_Frame_Go3)
  MoveL (TvRack_Frame_Go4)
  MoveL (TvRack_Frame_Fill)

--- program TvRack_Screen_ToFill (robot TvRack_Screen) ---
  Set Ref.: TvRack_Screen_Targets
  MoveL (TvRack_Screen_Go3)
  MoveL (TvRack_Screen_Go4)
  MoveL (TvRack_Screen_Fill)

--- Python program Reset_MainConveyor ---
# Type help("robolink") or help("robodk") for more information
# Press F5 to run the script
# Documentation: https://robodk.com/doc/en/RoboDK-API.html
# Reference:     https://robodk.com/doc/en/PythonAPI/index.html
# Note: It is not required to keep a copy of this file, your python script is saved with the station
from robodk import robolink
RDK = robolink.Robolink()


#---- Constant -----
NEW_REF_OBJECT_NAME = 'AssemblyRack_Ref' #Name of the ref object to copy
NEW_OBJECT_NAME = 'AssemblyRack' #Name of the new object created
REFERENCE_FRAME = 'MainConveyorRef' #Name of the frame the object will move to
REFERENCE_FRAME_REF = 'MainConveyorRef_Init'
MECHANISM_NAME = 'MainConveyor'

mechanism = RDK.Item(MECHANISM_NAME,itemtype=robolink.ITEM_TYPE_ROBOT)

#------- Program ------
frame = RDK.Item(REFERENCE_FRAME, robolink.ITEM_TYPE_FRAME)
frame_ref = RDK.Item(REFERENCE_FRAME_REF, robolink.ITEM_TYPE_FRAME)
ref_obj = RDK.Item(NEW_REF_OBJECT_NAME, robolink.ITEM_TYPE_OBJECT)


RDK.Render(False)

if mechanism.Valid():
    mechanism.setJoints([0])

if frame.Valid():
    for item in frame.Childs():
        if item.Type() == robolink.ITEM_TYPE_OBJECT:
            item.Delete()

for item in frame_ref.Childs():
    if frame.Valid() and  ref_obj.Valid():
        item.Copy()
        new_obj = RDK.Paste()
        new_obj.setVisible(False)
        new_obj.setParent(frame_ref)
        #new_obj.setName(NEW_OBJECT_NAME)
        RDK.Update()
        new_obj.setParentStatic(frame)
        new_obj.setVisible(True)

RDK.Render(True)

--- Python program Reset_Tool ---
# Type help("robolink") or help("robodk") for more information
# Press F5 to run the script
# Documentation: https://robodk.com/doc/en/RoboDK-API.html
# Reference:     https://robodk.com/doc/en/PythonAPI/index.html
# Note: It is not required to keep a copy of this file, your python script is saved with the station
from robolink import *    # RoboDK API
from robodk import *      # Robot toolbox
RDK2 = Robolink()

#----- CONSTANT -----

TOOL_NAME1 = 'ToolRobot1_TCP_Cup' #Name of the ref object to copy
TOOL_NAME2 = 'DeltaRobotTool' #Name of the ref object to copy
TOOL_NAME3 = 'ToolRobot1_TCP_Gripper' #Name of the ref object to copy
TOOL_NAME4 = 'TVAssemblyTCP' #Name of the ref object to copy
TOOL_NAME5 = 'AssemblyRackTCP' #Name of the ref object to copy
TOOL_NAME6 = 'ScrewTCP' #Name of the ref object to copy
TOOL_NAME7 = 'ToolRobot2TCP' #Name of the ref object to copy
TOOL_NAME8 = 'VaccumTool' #Name of the ref object to copy

#----- PROGRAM -----
tool1 = RDK2.Item(TOOL_NAME1,ITEM_TYPE_TOOL)
tool2 = RDK2.Item(TOOL_NAME2,ITEM_TYPE_TOOL)
tool3 = RDK2.Item(TOOL_NAME3,ITEM_TYPE_TOOL)
tool4 = RDK2.Item(TOOL_NAME4,ITEM_TYPE_TOOL)
tool5 = RDK2.Item(TOOL_NAME5,ITEM_TYPE_TOOL)
tool6 = RDK2.Item(TOOL_NAME6,ITEM_TYPE_TOOL)
tool7 = RDK2.Item(TOOL_NAME7,ITEM_TYPE_TOOL)
tool8 = RDK2.Item(TOOL_NAME8,ITEM_TYPE_TOOL)

if tool1.Valid():
    for item in tool1.Childs():
        if item.Type() == ITEM_TYPE_OBJECT:
            item.Delete()

if tool2.Valid():
    for item in tool2.Childs():
        if item.Type() == ITEM_TYPE_OBJECT:
            item.Delete()

if tool3.Valid():
    for item in tool3.Childs():
        if item.Type() == ITEM_TYPE_OBJECT:
            item.Delete()

if tool4.Valid():
    for item in tool4.Childs():
        if item.Type() == ITEM_TYPE_OBJECT:
            item.Delete()

if tool5.Valid():
    for item in tool5.Childs():
        if item.Type() == ITEM_TYPE_OBJECT:
            item.Delete()

if tool6.Valid():
    for item in tool6.Childs():
        if item.Type() == ITEM_TYPE_OBJECT:
            item.Delete()

if tool7.Valid():
    for item in tool7.Childs():
        if item.Type() == ITEM_TYPE_OBJECT:
            item.Delete()


if tool8.Valid():
    for item in tool8.Childs():
        if item.Type() == ITEM_TYPE_OBJECT:
            item.Delete()

--- Python program Reset_RackConveyor ---
# Type help("robolink") or help("robodk") for more information
# Press F5 to run the script
# Documentation: https://robodk.com/doc/en/RoboDK-API.html
# Reference:     https://robodk.com/doc/en/PythonAPI/index.html
# Note: It is not required to keep a copy of this file, your python script is saved with the station
from robodk import robolink
RDK = robolink.Robolink()

#----- Constant -----
NEW_REF_OBJECT_NAME = 'AssemblyRack_Ref' #Name of the ref object to copy
NEW_OBJECT_NAME = 'AssemblyRack' #Name of the new object created
REFERENCE_FRAME = 'AssemblyRackConveyorRef' #Name of the frame the object will move to
REFERENCE_FRAME_REF = 'AssemblyRackConveyorRef_Init'
MECHANISM_NAME = 'AssemblyRackConveyor'

mechanism = RDK.Item(MECHANISM_NAME,itemtype=robolink.ITEM_TYPE_ROBOT)

#------- Program ------
frame = RDK.Item(REFERENCE_FRAME, robolink.ITEM_TYPE_FRAME)
frame_ref = RDK.Item(REFERENCE_FRAME_REF, robolink.ITEM_TYPE_FRAME)
ref_obj = RDK.Item(NEW_REF_OBJECT_NAME, robolink.ITEM_TYPE_OBJECT)


RDK.Render(False)

if mechanism.Valid():
    mechanism.setJoints([0])

if frame.Valid():
    for item in frame.Childs():
        if item.Type() == robolink.ITEM_TYPE_OBJECT:
            item.Delete()



for item in frame_ref.Childs():
    if frame.Valid() and  ref_obj.Valid():
        item.Copy()
        new_obj = RDK.Paste()
        new_obj.setVisible(False)
        new_obj.setParent(frame_ref)
        RDK.Update()
        new_obj.setName(NEW_OBJECT_NAME)
        new_obj.setParentStatic(frame)
        new_obj.setVisible(True)

RDK.Render(True)

--- Python program Render ---
# Type help("robolink") or help("robodk") for more information
# Press F5 to run the script
# Documentation: https://robodk.com/doc/en/RoboDK-API.html
# Reference:     https://robodk.com/doc/en/PythonAPI/index.html
# Note: It is not required to keep a copy of this file, your python script is saved with the station
from robodk import robolink
RDK = robolink.Robolink()


RDK.Render(True)
RDK.Update()

--- Python program Reset_AVG ---
# Type help("robolink") or help("robodk") for more information
# Press F5 to run the script
# Documentation: https://robodk.com/doc/en/RoboDK-API.html
# Reference:     https://robodk.com/doc/en/PythonAPI/index.html
# Note: It is not required to keep a copy of this file, your python script is saved with the station
from robodk import robolink, robomath
RDK = robolink.Robolink()


#----- Constant -----
NEW_REF_OBJECT_NAME_TVFRAME = 'TVFrame_Ref' #Name of the ref object to copy
NEW_OBJECT_NAME_TVFRAME = 'TVFrame' #Name of the new object created
REFERENCE_FRAME_TVFRAME = 'TvRack_Frame_Ref' #Name of the frame the object will move to
REFERENCE_FRAME_REF_TVFRAME = 'TvRack_Frame_Init'
MECHANISM_NAME_TVFRAME = 'TvRack_Frame'


#----- Constant -----
NEW_REF_OBJECT_NAME_PANEL = 'TVFrontPanel_Ref' #Name of the ref object to copy
NEW_OBJECT_NAME_PANEL = 'TVFrontPanel' #Name of the new object created
REFERENCE_FRAME_PANEL = 'TvRack_FrontPanel_Ref' #Name of the frame the object will move to
REFERENCE_FRAME_REF_PANEL = 'TvRack_FrontPanel_Init'
MECHANISM_NAME_PANEL = 'TvRack_FrontPanel'


#----- Constant -----
NEW_REF_OBJECT_NAME_SCREEN = 'TVScreen_Ref' #Name of the ref object to copy
NEW_OBJECT_NAME_SCREEN = 'TVScreen' #Name of the new object created
REFERENCE_FRAME_SCREEN = 'TvRack_Screen_Ref' #Name of the frame the object will move to
REFERENCE_FRAME_REF_SCREEN = 'TvRack_Screen_Init'
MECHANISM_NAME_SCREEN = 'TvRack_Screen'



mechanism_tvframe = RDK.Item(MECHANISM_NAME_TVFRAME,itemtype=robolink.ITEM_TYPE_ROBOT)
mechanism_tvfrontpanel = RDK.Item(MECHANISM_NAME_PANEL,itemtype=robolink.ITEM_TYPE_ROBOT)
mechanism_tvscreen = RDK.Item(MECHANISM_NAME_SCREEN,itemtype=robolink.ITEM_TYPE_ROBOT)

#------- Program ------
frame_tvframe = RDK.Item(REFERENCE_FRAME_TVFRAME, robolink.ITEM_TYPE_FRAME)
frame_tvfrontpanel = RDK.Item(REFERENCE_FRAME_PANEL, robolink.ITEM_TYPE_FRAME)
frame_tvcreen = RDK.Item(REFERENCE_FRAME_SCREEN, robolink.ITEM_TYPE_FRAME)

frame_ref_tvframe = RDK.Item(REFERENCE_FRAME_REF_TVFRAME, robolink.ITEM_TYPE_FRAME)
frame_ref_tvfrontpanel = RDK.Item(REFERENCE_FRAME_REF_PANEL, robolink.ITEM_TYPE_FRAME)
frame_ref_tvscreen = RDK.Item(REFERENCE_FRAME_REF_SCREEN, robolink.ITEM_TYPE_FRAME)


ref_obj_tvframe = RDK.Item(NEW_OBJECT_NAME_TVFRAME, robolink.ITEM_TYPE_OBJECT)
ref_obj_tvfrontpanel = RDK.Item(NEW_OBJECT_NAME_PANEL, robolink.ITEM_TYPE_OBJECT)
ref_obj_tvscreen = RDK.Item(NEW_OBJECT_NAME_SCREEN, robolink.ITEM_TYPE_OBJECT)


RDK.Render(False)

if frame_tvframe.Valid():
    for item in frame_tvframe.Childs():
        if item.Type() == robolink.ITEM_TYPE_OBJECT:
            item.Delete()

if frame_tvfrontpanel.Valid():
    for item in frame_tvfrontpanel.Childs():
        if item.Type() == robolink.ITEM_TYPE_OBJECT:
            item.Delete()

if frame_tvcreen.Valid():
    for item in frame_tvcreen.Childs():
        if item.Type() == robolink.ITEM_TYPE_OBJECT:
            item.Delete()

if mechanism_tvframe.Valid():
    mechanism_tvframe.setJoints([-1600,-2100])

if mechanism_tvfrontpanel.Valid():
    mechanism_tvfrontpanel.setJoints([-710,-2100])

if mechanism_tvscreen.Valid():
    mechanism_tvscreen.setJoints([-2480,-2100])

for item in frame_ref_tvframe.Childs():
    if frame_tvframe.Valid() and  ref_obj_tvframe.Valid():
        item.Copy()
        new_obj = RDK.Paste()
        new_obj.setVisible(False)
        new_obj.setParent(frame_ref_tvframe)
        RDK.Update()
        new_obj.setName(NEW_OBJECT_NAME_TVFRAME)
        new_obj.setParentStatic(frame_tvframe)
        new_obj.setVisible(True)


for item in frame_ref_tvscreen.Childs():
    if frame_tvcreen.Valid() and  ref_obj_tvscreen.Valid():
        item.Copy()
        new_obj = RDK.Paste()
        new_obj.setVisible(False)
        new_obj.setParent(frame_ref_tvscreen)
        RDK.Update()
        new_obj.setName(NEW_OBJECT_NAME_SCREEN)
        new_obj.setParentStatic(frame_tvcreen)
        new_obj.setVisible(True)

for item in frame_ref_tvfrontpanel.Childs():
    if frame_tvfrontpanel.Valid() and  ref_obj_tvfrontpanel.Valid():
        item.Copy()
        new_obj = RDK.Paste()
        new_obj.setVisible(False)
        new_obj.setParent(frame_ref_tvfrontpanel)
        RDK.Update()
        new_obj.setName(NEW_OBJECT_NAME_PANEL)
        new_obj.setParentStatic(frame_tvfrontpanel)
        new_obj.setVisible(True)

RDK.Render(True)
RDK.Update()

--- Python program Reset_RackTargetRel ---
# Type help("robolink") or help("robodk") for more information
# Press F5 to run the script
# Documentation: https://robodk.com/doc/en/RoboDK-API.html
# Reference:     https://robodk.com/doc/en/PythonAPI/index.html
# Note: It is not required to keep a copy of this file, your python script is saved with the station
from robolink import *    # RoboDK API
from robodk import *      # Robot toolbox
RDK = Robolink()

#----- CONSTANT -----

#----- PROGRAM -----
TARGETscreen = 'RobotSFP_PickScreen'
TARGETframe = 'RobotSFP_PickFrame'
TARGETfrontpanel = 'RobotSFP_PickFrontPanel'
RDK.Render(False)

#----- PROGRAM -----
targetscreen = RDK.Item(TARGETscreen,ITEM_TYPE_TARGET)
targetfrontpanel = RDK.Item(TARGETfrontpanel,ITEM_TYPE_TARGET)
targetframe = RDK.Item(TARGETframe,ITEM_TYPE_TARGET)


targetscreen.setPose(Offset(targetscreen.Pose(),0,0,12))
targetfrontpanel.setPose(Offset(targetfrontpanel.Pose(),0,0,30))
targetframe.setPose(Offset(targetframe.Pose(),0,0,15))

RDK.Render(True)
RDK.Update()

--- Python program Reset_RackTargetABS ---
# Type help("robolink") or help("robodk") for more information
# Press F5 to run the script
# Documentation: https://robodk.com/doc/en/RoboDK-API.html
# Reference:     https://robodk.com/doc/en/PythonAPI/index.html
# Note: It is not required to keep a copy of this file, your python script is saved with the station
from robolink import *    # RoboDK API
from robodk import *      # Robot toolbox
RDK = Robolink()

#----- CONSTANT -----

TARGETscreen = 'RobotSFP_PickScreen'
TARGETframe = 'RobotSFP_PickFrame'
TARGETfrontpanel = 'RobotSFP_PickFrontPanel'

RDK.Render(False)

#----- PROGRAM -----
targetscreen = RDK.Item(TARGETscreen,ITEM_TYPE_TARGET)
targetfrontpanel = RDK.Item(TARGETfrontpanel,ITEM_TYPE_TARGET)
targetframe = RDK.Item(TARGETframe,ITEM_TYPE_TARGET)

x_screen=-3355.00
y_screen=320.00
z_screen=767.00

x_frontpanel=-3193.00
y_frontpanel=-1435.00
z_frontpanel=654.000

x_frame=-3200.00
y_frame=-555.00
z_frame=389.00


targetscreen.setPoseAbs(Pose(x_screen,y_screen,z_screen,0,-40,-90))
targetfrontpanel.setPoseAbs(Pose(x_frontpanel,y_frontpanel,z_frontpanel,0,-180,90))
targetframe.setPoseAbs(Pose(x_frame,y_frame,z_frame,0,-180,90))

RDK.Render(True)
RDK.Update()

--- program ResetALL (robot ABB IRB 2400/16) ---
  Call Reset_AVG
  Call Reset_BoxTargetABS
  Call Reset_RackConveyor
  Call Reset_Tool
  Call Reset_MainConveyor
  Call Reset_RackTargetABS
  Call Render

--- program Main (robot ABB IRB 2400/16) ---
  Call TvRack_ToPickUp
  Call TVAssembly_Main
  Call TVAssembly_Main
  Call TVAssembly_Main
  Call TvRack_BackToFill
  Call ResetALL
